(* PLC project Rasi_feeds_batching.project, Automation Builder 2.7 - Basic Automation Builder 2.7 *)
(* stored: creationDateTime 2026-08-29T13:50:00 *)

PROGRAM batching14
  VAR
    Auto_Ctrl : Auto_Batching_V14;
    Semi_Auto_Ctrl : Semi_Auto_Batching_V14;
    Auto_Complete : BOOL;
    Semi_Auto_Complete : BOOL;
    Auto_Err : INT;
    Semi_Auto_Err : INT;
  END_VAR

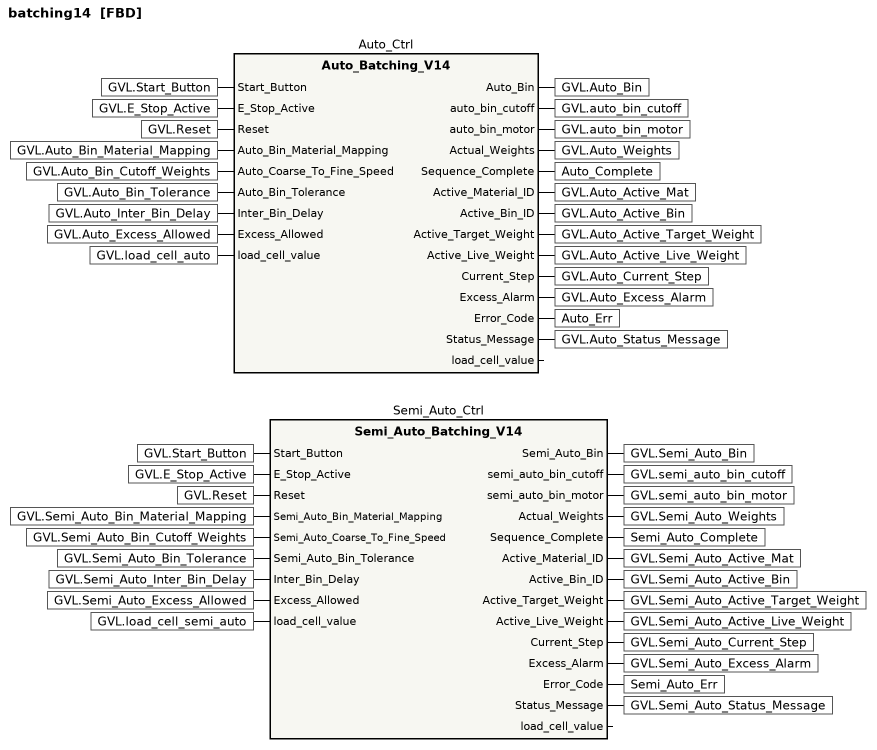
(* FBD diagram, written out as Structured Text *)
Auto_Ctrl(Start_Button := GVL.Start_Button, E_Stop_Active := GVL.E_Stop_Active, Reset := GVL.Reset, Auto_Bin_Material_Mapping := GVL.Auto_Bin_Material_Mapping, Auto_Coarse_To_Fine_Speed := GVL.Auto_Bin_Cutoff_Weights, Auto_Bin_Tolerance := GVL.Auto_Bin_Tolerance, Inter_Bin_Delay := GVL.Auto_Inter_Bin_Delay, Excess_Allowed := GVL.Auto_Excess_Allowed, load_cell_value := GVL.load_cell_auto);
GVL.Auto_Bin := Auto_Ctrl.Auto_Bin;
GVL.auto_bin_cutoff := Auto_Ctrl.auto_bin_cutoff;
GVL.auto_bin_motor := Auto_Ctrl.auto_bin_motor;
GVL.Auto_Weights := Auto_Ctrl.Actual_Weights;
Auto_Complete := Auto_Ctrl.Sequence_Complete;
GVL.Auto_Active_Mat := Auto_Ctrl.Active_Material_ID;
GVL.Auto_Active_Bin := Auto_Ctrl.Active_Bin_ID;
GVL.Auto_Active_Target_Weight := Auto_Ctrl.Active_Target_Weight;
GVL.Auto_Active_Live_Weight := Auto_Ctrl.Active_Live_Weight;
GVL.Auto_Current_Step := Auto_Ctrl.Current_Step;
GVL.Auto_Excess_Alarm := Auto_Ctrl.Excess_Alarm;
Auto_Err := Auto_Ctrl.Error_Code;
GVL.Auto_Status_Message := Auto_Ctrl.Status_Message;
Semi_Auto_Ctrl(Start_Button := GVL.Start_Button, E_Stop_Active := GVL.E_Stop_Active, Reset := GVL.Reset, Semi_Auto_Bin_Material_Mapping := GVL.Semi_Auto_Bin_Material_Mapping, Semi_Auto_Coarse_To_Fine_Speed := GVL.Semi_Auto_Bin_Cutoff_Weights, Semi_Auto_Bin_Tolerance := GVL.Semi_Auto_Bin_Tolerance, Inter_Bin_Delay := GVL.Semi_Auto_Inter_Bin_Delay, Excess_Allowed := GVL.Semi_Auto_Excess_Allowed, load_cell_value := GVL.load_cell_semi_auto);
GVL.Semi_Auto_Bin := Semi_Auto_Ctrl.Semi_Auto_Bin;
GVL.semi_auto_bin_cutoff := Semi_Auto_Ctrl.semi_auto_bin_cutoff;
GVL.semi_auto_bin_motor := Semi_Auto_Ctrl.semi_auto_bin_motor;
GVL.Semi_Auto_Weights := Semi_Auto_Ctrl.Actual_Weights;
Semi_Auto_Complete := Semi_Auto_Ctrl.Sequence_Complete;
GVL.Semi_Auto_Active_Mat := Semi_Auto_Ctrl.Active_Material_ID;
GVL.Semi_Auto_Active_Bin := Semi_Auto_Ctrl.Active_Bin_ID;
GVL.Semi_Auto_Active_Target_Weight := Semi_Auto_Ctrl.Active_Target_Weight;
GVL.Semi_Auto_Active_Live_Weight := Semi_Auto_Ctrl.Active_Live_Weight;
GVL.Semi_Auto_Current_Step := Semi_Auto_Ctrl.Current_Step;
GVL.Semi_Auto_Excess_Alarm := Semi_Auto_Ctrl.Excess_Alarm;
Semi_Auto_Err := Semi_Auto_Ctrl.Error_Code;
GVL.Semi_Auto_Status_Message := Semi_Auto_Ctrl.Status_Message;
END_PROGRAM
